(* ================================================================= *)
(*  FB_1012_ConveyorMotor                                             *)
(*  输送电机控制 - 方向仲裁+安全门互锁+VFD故障检测                    *)
(*  版本: V8.0.0  日期: 2026-05-27                                    *)
(*  来源: SysLib/actuator/                                            *)
(*  规范: 801_DEV-V1.0.5, 810_DEV-V1.0.2                             *)
(*                                                                    *)
(*  V8.0.0变更:                                                       *)
(*    - 重构: 扁平化VAR_INPUT/OUTPUT → VAR_IN_OUT ST_ConveyorMotor    *)
(*    - 对齐: 命令/安全/参数/输出/状态全部通过ST_ConveyorMotor结构体  *)
(*    - 参考: FB_1003 VAR_IN_OUT io_stZAxis:ST_ServoAxis 模式        *)
(* ================================================================= *)

FUNCTION_BLOCK FB_1012_ConveyorMotor

VAR_INPUT
END_VAR

VAR_OUTPUT
END_VAR

VAR_IN_OUT
    io_stMotor      : ST_ConveyorMotor; (* 电机结构体: 命令/安全/参数/输出/状态 *)
END_VAR

(* ==================== VFD故障检测 最高优先级 ==================== *)
IF io_stMotor.VfdFault THEN
    io_stMotor.VfdAlarm := TRUE;
    io_stMotor.FwdOut := FALSE;
    io_stMotor.RevOut := FALSE;
    io_stMotor.SlowOut := FALSE;
    io_stMotor.Running := FALSE;
    RETURN;
ELSE
    io_stMotor.VfdAlarm := FALSE;
END_IF;

(* ==================== 安全门互锁 ==================== *)
IF NOT io_stMotor.SafetyDoorOk THEN
    io_stMotor.FwdOut := FALSE;
    io_stMotor.RevOut := FALSE;
    io_stMotor.SlowOut := FALSE;
    io_stMotor.Running := FALSE;
    RETURN;
END_IF;

(* ==================== 方向命令仲裁 Fwd > Rev > Slow ==================== *)
IF io_stMotor.FwdCmd THEN
    io_stMotor.FwdOut := TRUE;
    io_stMotor.RevOut := FALSE;
    io_stMotor.SlowOut := FALSE;
    io_stMotor.Running := TRUE;
ELSIF io_stMotor.RevCmd THEN
    io_stMotor.FwdOut := FALSE;
    io_stMotor.RevOut := TRUE;
    io_stMotor.SlowOut := FALSE;
    io_stMotor.Running := TRUE;
ELSIF io_stMotor.SlowCmd THEN
    io_stMotor.FwdOut := FALSE;
    io_stMotor.RevOut := FALSE;
    io_stMotor.SlowOut := TRUE;
    io_stMotor.Running := TRUE;
ELSE
    io_stMotor.FwdOut := FALSE;
    io_stMotor.RevOut := FALSE;
    io_stMotor.SlowOut := FALSE;
    io_stMotor.Running := FALSE;
END_IF;

END_FUNCTION_BLOCK
